// LS Electric XG5000 project: Twin color_1200IMM
// PLC NewPLC
// module base 0 slot 0: Input/Output Module:XBC-DR28U (DC 24V INPUT 16points/RELAY OUTPUT 12points)
// module base 0 slot 1: Embedded Analog IO :XBF-AH8E (Input 4CH, Current Output 2CH, Voltage Output 2CH)
// module base 0 slot 2: Temp. Measuring Module:XBF-TC04S (TC, 4-CH)

PROGRAM NewProgram (task: Scan Program)

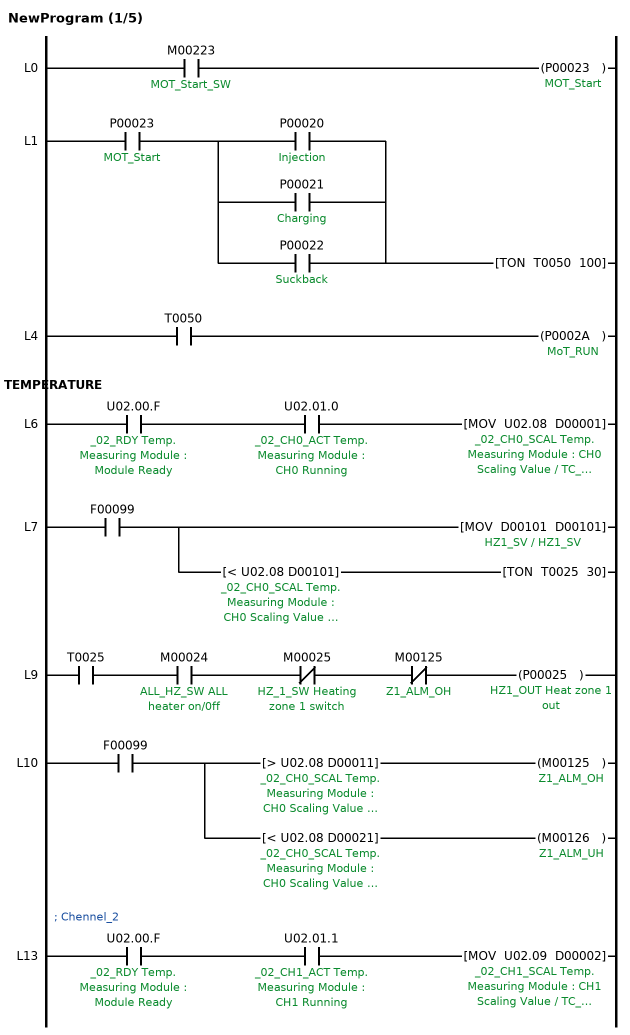
; L0
LOAD      M00223	// MOT_Start_SW
OUT       P00023	// MOT_Start
; L1
LOAD      P00023	// MOT_Start
LOAD      P00020	// Injection
OR        P00021	// Charging
OR        P00022	// Suckback
AND LOAD
TON       T0050 100
; L4
LOAD      T0050
OUT       P0002A	// MoT_RUN
TEMPERATURE:
; L6
LOAD      U02.00.F	// _02_RDY Temp. Measuring Module : Module Ready
AND       U02.01.0	// _02_CH0_ACT Temp. Measuring Module : CH0 Running
MOV       U02.08 D00001	// _02_CH0_SCAL Temp. Measuring Module : CH0 Scaling Value / TC_1 Temp.Zone 1 thermocouple input
; L7
LOAD      F00099
MOV       D00101 D00101	// HZ1_SV / HZ1_SV
AND<      U02.08 D00101	// _02_CH0_SCAL Temp. Measuring Module : CH0 Scaling Value / HZ1_SV
TON       T0025 30
; L9
LOAD      T0025
AND       M00024	// ALL_HZ_SW ALL heater on/0ff
AND NOT   M00025	// HZ_1_SW Heating zone 1 switch
AND NOT   M00125	// Z1_ALM_OH
OUT       P00025	// HZ1_OUT Heat zone 1 out
; L10
LOAD      F00099
MPUSH
AND>      U02.08 D00011	// _02_CH0_SCAL Temp. Measuring Module : CH0 Scaling Value / MSV_Z1
OUT       M00125	// Z1_ALM_OH
MPOP
AND<      U02.08 D00021	// _02_CH0_SCAL Temp. Measuring Module : CH0 Scaling Value / LSV_Z1 Lower value zone 1
OUT       M00126	// Z1_ALM_UH
// Chennel_2
; L13
LOAD      U02.00.F	// _02_RDY Temp. Measuring Module : Module Ready
AND       U02.01.1	// _02_CH1_ACT Temp. Measuring Module : CH1 Running
MOV       U02.09 D00002	// _02_CH1_SCAL Temp. Measuring Module : CH1 Scaling Value / TC_2 Temp.Zone 1 thermocouple input

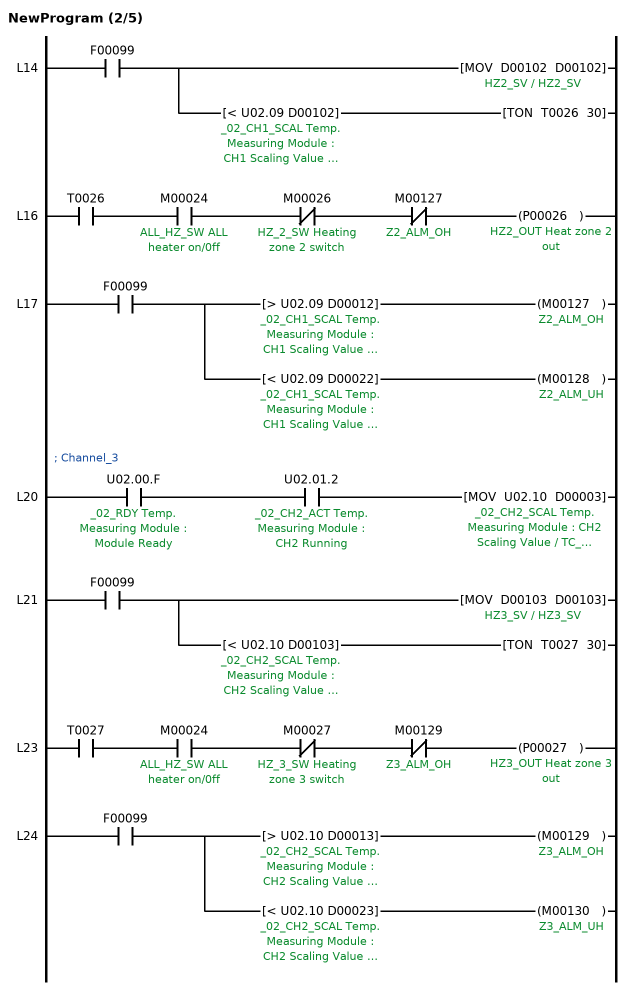
; L14
LOAD      F00099
MOV       D00102 D00102	// HZ2_SV / HZ2_SV
AND<      U02.09 D00102	// _02_CH1_SCAL Temp. Measuring Module : CH1 Scaling Value / HZ2_SV
TON       T0026 30
; L16
LOAD      T0026
AND       M00024	// ALL_HZ_SW ALL heater on/0ff
AND NOT   M00026	// HZ_2_SW Heating zone 2 switch
AND NOT   M00127	// Z2_ALM_OH
OUT       P00026	// HZ2_OUT Heat zone 2 out
; L17
LOAD      F00099
MPUSH
AND>      U02.09 D00012	// _02_CH1_SCAL Temp. Measuring Module : CH1 Scaling Value / MSV_Z2
OUT       M00127	// Z2_ALM_OH
MPOP
AND<      U02.09 D00022	// _02_CH1_SCAL Temp. Measuring Module : CH1 Scaling Value / LSV_Z2
OUT       M00128	// Z2_ALM_UH
// Channel_3
; L20
LOAD      U02.00.F	// _02_RDY Temp. Measuring Module : Module Ready
AND       U02.01.2	// _02_CH2_ACT Temp. Measuring Module : CH2 Running
MOV       U02.10 D00003	// _02_CH2_SCAL Temp. Measuring Module : CH2 Scaling Value / TC_3 Temp.Zone 1 thermocouple input
; L21
LOAD      F00099
MOV       D00103 D00103	// HZ3_SV / HZ3_SV
AND<      U02.10 D00103	// _02_CH2_SCAL Temp. Measuring Module : CH2 Scaling Value / HZ3_SV
TON       T0027 30
; L23
LOAD      T0027
AND       M00024	// ALL_HZ_SW ALL heater on/0ff
AND NOT   M00027	// HZ_3_SW Heating zone 3 switch
AND NOT   M00129	// Z3_ALM_OH
OUT       P00027	// HZ3_OUT Heat zone 3 out
; L24
LOAD      F00099
MPUSH
AND>      U02.10 D00013	// _02_CH2_SCAL Temp. Measuring Module : CH2 Scaling Value / MSV_Z3
OUT       M00129	// Z3_ALM_OH
MPOP
AND<      U02.10 D00023	// _02_CH2_SCAL Temp. Measuring Module : CH2 Scaling Value / LSV_Z3
OUT       M00130	// Z3_ALM_UH

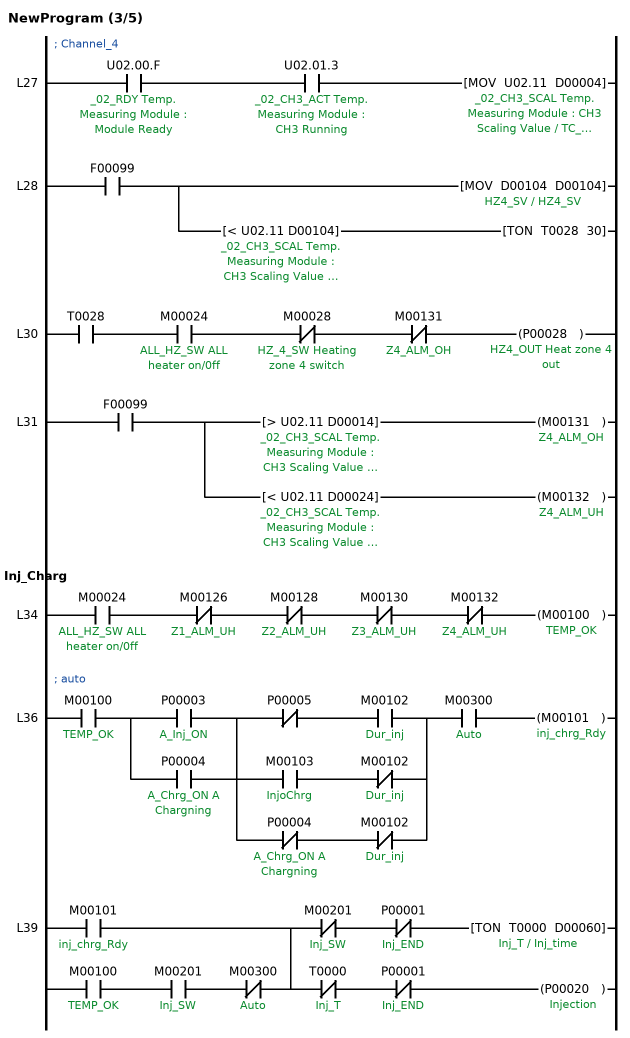
// Channel_4
; L27
LOAD      U02.00.F	// _02_RDY Temp. Measuring Module : Module Ready
AND       U02.01.3	// _02_CH3_ACT Temp. Measuring Module : CH3 Running
MOV       U02.11 D00004	// _02_CH3_SCAL Temp. Measuring Module : CH3 Scaling Value / TC_4 Temp.Zone 1 thermocouple input
; L28
LOAD      F00099
MOV       D00104 D00104	// HZ4_SV / HZ4_SV
AND<      U02.11 D00104	// _02_CH3_SCAL Temp. Measuring Module : CH3 Scaling Value / HZ4_SV
TON       T0028 30
; L30
LOAD      T0028
AND       M00024	// ALL_HZ_SW ALL heater on/0ff
AND NOT   M00028	// HZ_4_SW Heating zone 4 switch
AND NOT   M00131	// Z4_ALM_OH
OUT       P00028	// HZ4_OUT Heat zone 4 out
; L31
LOAD      F00099
MPUSH
AND>      U02.11 D00014	// _02_CH3_SCAL Temp. Measuring Module : CH3 Scaling Value / MSV_Z4
OUT       M00131	// Z4_ALM_OH
MPOP
AND<      U02.11 D00024	// _02_CH3_SCAL Temp. Measuring Module : CH3 Scaling Value / LSV_Z4
OUT       M00132	// Z4_ALM_UH
Inj_Charg:
; L34
LOAD      M00024	// ALL_HZ_SW ALL heater on/0ff
AND NOT   M00126	// Z1_ALM_UH
AND NOT   M00128	// Z2_ALM_UH
AND NOT   M00130	// Z3_ALM_UH
AND NOT   M00132	// Z4_ALM_UH
OUT       M00100	// TEMP_OK
// auto
; L36
LOAD      M00100	// TEMP_OK
LOAD      P00003	// A_Inj_ON
OR        P00004	// A_Chrg_ON A Chargning
AND LOAD
LOAD NOT  P00005
AND       M00102	// Dur_inj
LOAD      M00103	// InjoChrg
AND NOT   M00102	// Dur_inj
OR LOAD
LOAD NOT  P00004	// A_Chrg_ON A Chargning
AND NOT   M00102	// Dur_inj
OR LOAD
AND LOAD
AND       M00300	// Auto
OUT       M00101	// inj_chrg_Rdy
; L39
LOAD      M00101	// inj_chrg_Rdy
LOAD      M00100	// TEMP_OK
AND       M00201	// Inj_SW
AND NOT   M00300	// Auto
OR LOAD
MPUSH
AND NOT   M00201	// Inj_SW
AND NOT   P00001	// Inj_END
TON       T0000 D00060	// Inj_T / Inj_time
MPOP
AND NOT   T0000	// Inj_T
AND NOT   P00001	// Inj_END
OUT       P00020	// Injection

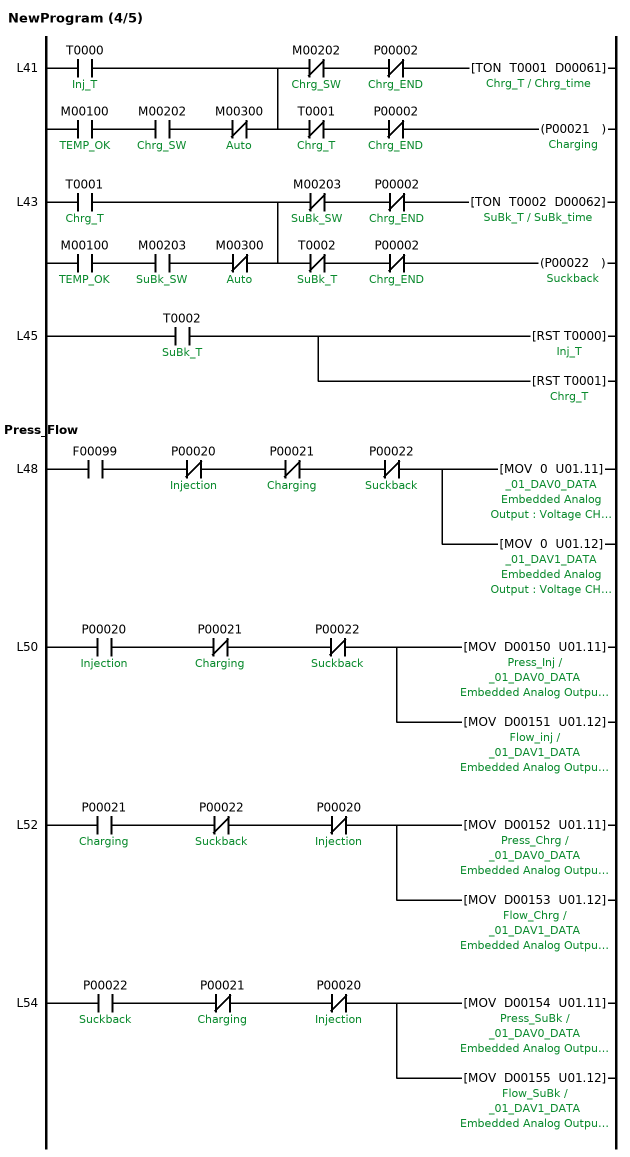
; L41
LOAD      T0000	// Inj_T
LOAD      M00100	// TEMP_OK
AND       M00202	// Chrg_SW
AND NOT   M00300	// Auto
OR LOAD
MPUSH
AND NOT   M00202	// Chrg_SW
AND NOT   P00002	// Chrg_END
TON       T0001 D00061	// Chrg_T / Chrg_time
MPOP
AND NOT   T0001	// Chrg_T
AND NOT   P00002	// Chrg_END
OUT       P00021	// Charging
; L43
LOAD      T0001	// Chrg_T
LOAD      M00100	// TEMP_OK
AND       M00203	// SuBk_SW
AND NOT   M00300	// Auto
OR LOAD
MPUSH
AND NOT   M00203	// SuBk_SW
AND NOT   P00002	// Chrg_END
TON       T0002 D00062	// SuBk_T / SuBk_time
MPOP
AND NOT   T0002	// SuBk_T
AND NOT   P00002	// Chrg_END
OUT       P00022	// Suckback
; L45
LOAD      T0002	// SuBk_T
RST       T0000	// Inj_T
RST       T0001	// Chrg_T
Press_Flow:
; L48
LOAD      F00099
AND NOT   P00020	// Injection
AND NOT   P00021	// Charging
AND NOT   P00022	// Suckback
MOV       0 U01.11	// _01_DAV0_DATA Embedded Analog Output : Voltage CH0 Input
MOV       0 U01.12	// _01_DAV1_DATA Embedded Analog Output : Voltage CH1 Input
; L50
LOAD      P00020	// Injection
AND NOT   P00021	// Charging
AND NOT   P00022	// Suckback
MOV       D00150 U01.11	// Press_Inj / _01_DAV0_DATA Embedded Analog Output : Voltage CH0 Input
MOV       D00151 U01.12	// Flow_inj / _01_DAV1_DATA Embedded Analog Output : Voltage CH1 Input
; L52
LOAD      P00021	// Charging
AND NOT   P00022	// Suckback
AND NOT   P00020	// Injection
MOV       D00152 U01.11	// Press_Chrg / _01_DAV0_DATA Embedded Analog Output : Voltage CH0 Input
MOV       D00153 U01.12	// Flow_Chrg / _01_DAV1_DATA Embedded Analog Output : Voltage CH1 Input
; L54
LOAD      P00022	// Suckback
AND NOT   P00021	// Charging
AND NOT   P00020	// Injection
MOV       D00154 U01.11	// Press_SuBk / _01_DAV0_DATA Embedded Analog Output : Voltage CH0 Input
MOV       D00155 U01.12	// Flow_SuBk / _01_DAV1_DATA Embedded Analog Output : Voltage CH1 Input

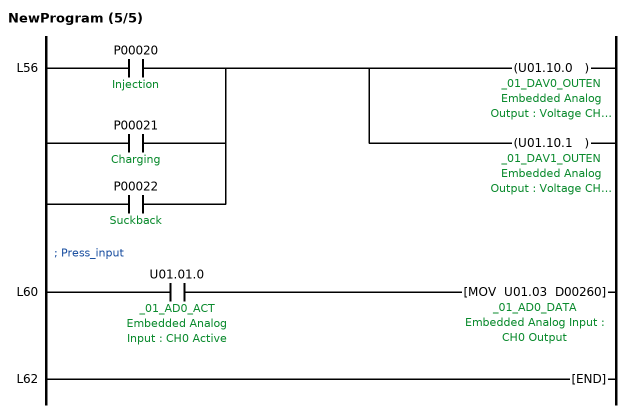
; L56
LOAD      P00020	// Injection
OR        P00021	// Charging
OR        P00022	// Suckback
OUT       U01.10.0	// _01_DAV0_OUTEN Embedded Analog Output : Voltage CH0 Output Status Setting
OUT       U01.10.1	// _01_DAV1_OUTEN Embedded Analog Output : Voltage CH1 Output Status Setting
// Press_input
; L60
LOAD      U01.01.0	// _01_AD0_ACT Embedded Analog Input : CH0 Active
MOV       U01.03 D00260	// _01_AD0_DATA Embedded Analog Input : CH0 Output
; L62
END

VARIABLES AND COMMENTS (devices not used above)
D00050	WORD	Inj_Dly
D00111	WORD	MV_1